TYPE ST_Component_TE2_HMI :
STRUCT
	bZmienneTypoweDlaComponent_TE2	: BOOL;
	
END_STRUCT
END_TYPE

(* stored: Version 1.1.0.1, ProductVersion 3.1.4024.15
   DUT ST_Component_TE2_HMI: Id {c5a187ad-86dc-432f-b19d-3e27f16be75b} *)
